PROGRAM MAIN
VAR
	
	CRAHs : AllCRAHs;
	
	ModbusComms: ModbusRTU;
END_VAR

ModbusComms();

CRAHs();

END_PROGRAM

(* stored: Version 1.1.0.1, ProductVersion 3.1.4024.12
   POU MAIN: Id {8dbe3832-cff4-4323-b62f-00c235c99abe}, SpecialFunc None *)
